// TIA Portal V19 export
DATA_BLOCK "FB_DEBUG_MES_DB"   // DB178
// stored: InstanceOfName FB_DEBUG_MES, InstanceOfType FB
"FB_DEBUG_MES"
   // VAR
   //    i : Int;
   //    CodiceAllarmePARTS { S7_SetPoint := 'True'} : Int;
   //    CodiceAllarmeBEAMS { S7_SetPoint := 'True'} : Int;
   //    R_TRIG_Deroga { S7_SetPoint := 'True'} : R_TRIG;
   //    R_TRIG_Provino_Eseguito { S7_SetPoint := 'True'} : R_TRIG;
   //    R_TRIG_SetUp_PartProd_Done { S7_SetPoint := 'True'} : R_TRIG;
   //    R_TRIG_SetUp_BeamProd_Done { S7_SetPoint := 'True'} : R_TRIG;
   //    R_TRIG_NewPart { S7_SetPoint := 'True'} : R_TRIG;
   //    R_TRIG_NewBeam { S7_SetPoint := 'True'} : R_TRIG;
   //    R_TRIG_TaglioLamiera { S7_SetPoint := 'True'} : R_TRIG;
   //    R_TRIG_Giunzione { S7_SetPoint := 'True'} : R_TRIG;
   //    R_TRIG_Giunzione_Dopo_Taglio_Finale { S7_SetPoint := 'True'} : R_TRIG;
   //    R_TRIG_Step_Introduzione { S7_SetPoint := 'True'} : R_TRIG;
   //    R_TRIG_Step_Vuotamento { S7_SetPoint := 'True'} : R_TRIG;
   //    R_TRIG_SimulaAllarmePARTS { S7_SetPoint := 'True'} : R_TRIG;
   //    R_TRIG_SimulaAllarmeBEAMS { S7_SetPoint := 'True'} : R_TRIG;
   //    R_TRIG_AutomaticoPARTS { S7_SetPoint := 'True'} : R_TRIG;
   //    R_TRIG_AutomaticoBEAMS { S7_SetPoint := 'True'} : R_TRIG;
   //    R_TRIG_PausaPARTS { S7_SetPoint := 'True'} : R_TRIG;
   //    R_TRIG_PausaBEAMS_2 { S7_SetPoint := 'True'} : R_TRIG;
   //    R_TRIG_PausaBEAMS_1 { S7_SetPoint := 'True'} : R_TRIG;
   //    R_TRIG_CambioAspo { S7_SetPoint := 'True'} : R_TRIG;
   //    CumulativoAllarmiProduzionePart { S7_SetPoint := 'True'} : Bool;
   //    CumulativoAllarmiProduzioneBeams { S7_SetPoint := 'True'} : Bool;
   //    WarningNoBeamsToHandle : Bool;
   //    R_TRIG_ResetStops { S7_SetPoint := 'True'} : R_TRIG;
   //    RETVAL_GetOrderData_O_ENDING { S7_SetPoint := 'True'} : DInt;
   //    Sel_ProdEndingIndx : Int;
   //    RETVAL_GetOrderData_O_ACT { S7_SetPoint := 'True'} : DInt;
   //    Sel_Free : Int;
   //    Ordine_Trovato : Bool;
   //    R_TRIG_MuoveSuBaiaDiUscita { S7_SetPoint := 'True'} : R_TRIG;
   //    RETVAL_INT { S7_SetPoint := 'True'} : Int;
   //    RETVAL_GetOrderData_Stacker { S7_SetPoint := 'True'} : DInt;
   //    Stacker_Order : "Prod_Item";
   //    Stacker_Index_O_Ending { S7_SetPoint := 'True'} : Int;
   // END_VAR
BEGIN
END_DATA_BLOCK
